(* PLC project Unbenannt, Unbekannt Unbenannt 1 *)
(* stored: creationDateTime 2019-08-31T23:44:27, modificationDateTime 2019-09-19T22:19:56 *)

(* BYTE_TO_STRINGH converts a Byte to a String of Hexadecimal represented by '0' .. '9' and 'A' .. 'F'. The lowest order Character will be on the right and the high order Character on the left. *)
FUNCTION_BLOCK BYTE_TO_STRH
  VAR_INPUT
    IN : BYTE;
  END_VAR
  VAR_OUTPUT
    _BYTE_TO_STRH : STRING;
  END_VAR
  VAR
    x : INT;
    c : BYTE;
    temp : STRING := '2';
    temp2 : BYTE;
  END_VAR

            _BYTE_TO_STRH:=BYTE_TO_STRING(IN,'%02X');







(* From Oscat Library, www.oscat.de *)
          
END_FUNCTION_BLOCK

PROGRAM program0
  VAR
    LocalVar0 : DINT;
    LocalVar1 : DINT;
    LocalVar2 : DINT;
  END_VAR

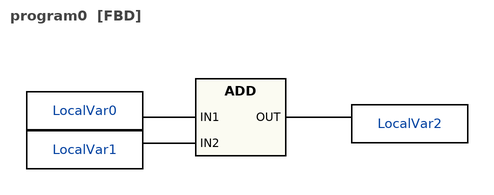
(* FBD diagram, written out as Structured Text *)
LocalVar2 := LocalVar0 + LocalVar1;
END_PROGRAM

FUNCTION_BLOCK BYTE_TO_STRB
  VAR_INPUT
    IN : BYTE;
    _BYTE_TO_STRB : STRING;
  END_VAR
  VAR
    i : INT;
  END_VAR

            _BYTE_TO_STRB := '';
FOR i := 1 TO 8 DO
    IF (in AND BYTE#2#1000_0000) = BYTE#2#1000_0000 THEN
        _BYTE_TO_STRB := CONCAT(_BYTE_TO_STRB,'1');
    ELSE
        _BYTE_TO_STRB := CONCAT(_BYTE_TO_STRB,'0');
    END_IF;
	in := SHL(in, 1);
END_FOR;

(* From Oscat Library, www.oscat.de *)
          
END_FUNCTION_BLOCK

CONFIGURATION Config0
  RESOURCE Res0 ON PLC
    TASK task0(INTERVAL := T#20ms, PRIORITY := 0);
    PROGRAM instance0 WITH task0 : program0;
  END_RESOURCE
END_CONFIGURATION
